PROGRAM prgComEffIO
VAR
	fbCom		: FB_MqttCommunicator_v3;

END_VAR

fbCom(
	bConnect:= TRUE, 
	strAuthkey := 'DEV01673741737',
	sUserName:= '0a132640-f2fb-4f7a-ac17-2fdb23c06541' , 		
	sUserPassword:= 'd65348be-07b8-4dac-9fba-07c06f3e7cbb',
	eSavePositionCertificate:= eSavePositionOnPLC.ePostionC, 
	bConnected=> , 
	bError=> , 
	hrErrorCode=> , 
	eConnectionState=> , 
	eErrorMessage_Out=> );

END_PROGRAM

(* stored: Version 1.1.0.1, ProductVersion 3.1.4024.12
   POU prgComEffIO: Id {7bcbbbc3-1bb8-41a4-b832-244390633677}, SpecialFunc None *)
